(* Logix 5000 project; controller RSL5k_18_Template_noLib Emulate 5570 rev 32.11; software revision 32.02; part 15 of 16 *)
(* tags used below, declared in another part *)
   L_TaskMonitor : L_TaskMon[8];

        [450].Desc := 'Two Phases Lost In Power Cell #22', [451].Code := 351, [451].Desc := 'Bypass Failure (OV) In Power Cell #22', [452].Code := 353, [452].Desc := 'IGBT Over Current In Power Cell #23', [453].Code := 354, [453].Desc := 'Capacitor Abnormal In Power Cell #23', [454].Code := 355, [454].Desc := 'Input Over Voltage In Power Cell #23', [455].Code := 356, [455].Desc := 'DC Bus Undervoltage In Power Cell #23', [456].Code := 357, [456].Desc := 'Communication Error In Power Cell #23', [457].Code := 358, [457].Desc := 'No PWM Pulse For IGBT In Power Cell #23', [458].Code := 359, [458].Desc := 'Bypass Hardware Fault In Power Cell #23', [459].Code := 360, [459].Desc := 'Comm Link Fault in Power Cell #23', [460].Code := 361, [460].Desc := 'PCCB Ver. Incompatible In Power Cell #23', [461].Code := 362, [461].Desc := 'Power Cell #23 Bypassed', [462].Code := 363, [462].Desc := 'Over Temperature In Power Cell #23', [463].Code := 364, [463].Desc := 'Power Cell #23 Failed To Bypass', [464].Code := 365, [464].Desc := 'One Phase Lost In Power Cell #23', [465].Code := 366, [465].Desc := 'Two Phases Lost In Power Cell #23', [466].Code := 367, [466].Desc := 'Bypass Failure (OV) In Power Cell #23', [467].Code := 369, [467].Desc := 'IGBT Over Current In Power Cell #24', [468].Code := 370, [468].Desc := 'Capacitor Abnormal In Power Cell #24', [469].Code := 371, [469].Desc := 'Input Over Voltage In Power Cell #24', [470].Code := 372, [470].Desc := 'DC Bus Undervoltage In Power Cell #24', [471].Code := 373, [471].Desc := 'Communication Error In Power Cell #24', [472].Code := 374, [472].Desc := 'No PWM Pulse For IGBT In Power Cell #24', [473].Code := 375, [473].Desc := 'Bypass Hardware Fault In Power Cell #24', [474].Code := 376, [474].Desc := 'Comm Link Fault in Power Cell #24', [475].Code := 377, [475].Desc := 'PCCB Ver. Incompatible In Power Cell #24', [476].Code := 378, [476].Desc := 'Power Cell #24 Bypassed', [477].Code := 379, [477].Desc := 'Over Temperature In Power Cell #24', [478].Code := 380, [478].Desc := 'Power Cell #24 Failed To Bypass', [479].Code := 381, [479].Desc := 'One Phase Lost In Power Cell #24', [480].Code := 382,
        [480].Desc := 'Two Phases Lost In Power Cell #24', [481].Code := 383, [481].Desc := 'Bypass Failure (OV) In Power Cell #24', [482].Code := 385, [482].Desc := 'IGBT Over Current In Power Cell #25', [483].Code := 386, [483].Desc := 'Capacitor Abnormal In Power Cell #25', [484].Code := 387, [484].Desc := 'Input Over Voltage In Power Cell #25', [485].Code := 388, [485].Desc := 'DC Bus Undervoltage In Power Cell #25', [486].Code := 389, [486].Desc := 'Communication Error In Power Cell #25', [487].Code := 390, [487].Desc := 'No PWM Pulse For IGBT In Power Cell #25', [488].Code := 391, [488].Desc := 'Bypass Hardware Fault In Power Cell #25', [489].Code := 392, [489].Desc := 'Comm Link Fault in Power Cell #25', [490].Code := 393, [490].Desc := 'PCCB Ver. Incompatible In Power Cell #25', [491].Code := 394, [491].Desc := 'Power Cell #25 Bypassed', [492].Code := 395, [492].Desc := 'Over Temperature In Power Cell #25', [493].Code := 396, [493].Desc := 'Power Cell #25 Failed To Bypass', [494].Code := 397, [494].Desc := 'One Phase Lost In Power Cell #25', [495].Code := 398, [495].Desc := 'Two Phases Lost In Power Cell #25', [496].Code := 399, [496].Desc := 'Bypass Failure (OV) In Power Cell #25', [497].Code := 401, [497].Desc := 'IGBT Over Current In Power Cell #26', [498].Code := 402, [498].Desc := 'Capacitor Abnormal In Power Cell #26', [499].Code := 403, [499].Desc := 'Input Over Voltage In Power Cell #26', [500].Code := 404, [500].Desc := 'DC Bus Undervoltage In Power Cell #26', [501].Code := 405, [501].Desc := 'Communication Error In Power Cell #26', [502].Code := 406, [502].Desc := 'No PWM Pulse For IGBT In Power Cell #26', [503].Code := 407, [503].Desc := 'Bypass Hardware Fault In Power Cell #26', [504].Code := 408, [504].Desc := 'Comm Link Fault in Power Cell #26', [505].Code := 409, [505].Desc := 'PCCB Ver. Incompatible In Power Cell #26', [506].Code := 410, [506].Desc := 'Power Cell #26 Bypassed', [507].Code := 411, [507].Desc := 'Over Temperature In Power Cell #26', [508].Code := 412, [508].Desc := 'Power Cell #26 Failed To Bypass', [509].Code := 413, [509].Desc := 'One Phase Lost In Power Cell #26', [510].Code := 414,
        [510].Desc := 'Two Phases Lost In Power Cell #26', [511].Code := 415, [511].Desc := 'Bypass Failure (OV) In Power Cell #26', [512].Code := 417, [512].Desc := 'IGBT Over Current In Power Cell #27', [513].Code := 418, [513].Desc := 'Capacitor Abnormal In Power Cell #27', [514].Code := 419, [514].Desc := 'Input Over Voltage In Power Cell #27', [515].Code := 420, [515].Desc := 'DC Bus Undervoltage In Power Cell #27', [516].Code := 421, [516].Desc := 'Communication Error In Power Cell #27', [517].Code := 422, [517].Desc := 'No PWM Pulse For IGBT In Power Cell #27', [518].Code := 423, [518].Desc := 'Bypass Hardware Fault In Power Cell #27', [519].Code := 424, [519].Desc := 'Comm Link Fault in Power Cell #27', [520].Code := 425, [520].Desc := 'PCCB Ver. Incompatible In Power Cell #27', [521].Code := 426, [521].Desc := 'Power Cell #27 Bypassed', [522].Code := 427, [522].Desc := 'Over Temperature In Power Cell #27', [523].Code := 428, [523].Desc := 'Power Cell #27 Failed To Bypass', [524].Code := 429, [524].Desc := 'One Phase Lost In Power Cell #27', [525].Code := 430, [525].Desc := 'Two Phases Lost In Power Cell #27', [526].Code := 431, [526].Desc := 'Bypass Failure (OV) In Power Cell #27', [527].Code := 497, [527].Desc := 'PWMA Board Not Compatible With PCCBA1', [528].Code := 498, [528].Desc := 'PWMA Board Not Compatible With PCCBA2', [529].Code := 499, [529].Desc := 'PWMA Board Not Compatible With PCCBA3', [530].Code := 500, [530].Desc := 'PWMA Board Not Compatible With PCCBA4', [531].Code := 501, [531].Desc := 'PWMA Board Not Compatible With PCCBA5', [532].Code := 502, [532].Desc := 'PWMA Board Not Compatible With PCCBA6', [533].Code := 503, [533].Desc := 'PWMA Board Not Compatible With PCCBA7', [534].Code := 504, [534].Desc := 'PWMA Board Not Compatible With PCCBA8', [535].Code := 505, [535].Desc := 'PWMA Board Not Compatible With PCCBA9', [536].Code := 513, [536].Desc := 'PWMB Board Not Compatible With PCCBB1', [537].Code := 514, [537].Desc := 'PWMB Board Not Compatible With PCCBB2', [538].Code := 515, [538].Desc := 'PWMB Board Not Compatible With PCCBB3', [539].Code := 516, [539].Desc := 'PWMB Board Not Compatible With PCCBB4', [540].Code := 517,
        [540].Desc := 'PWMB Board Not Compatible With PCCBB5', [541].Code := 518, [541].Desc := 'PWMB Board Not Compatible With PCCBB6', [542].Code := 519, [542].Desc := 'PWMB Board Not Compatible With PCCBB7', [543].Code := 520, [543].Desc := 'PWMB Board Not Compatible With PCCBB8', [544].Code := 521, [544].Desc := 'PWMB Board Not Compatible With PCCBB9', [545].Code := 529, [545].Desc := 'PWMC Board Not Compatible With PCCBC1', [546].Code := 530, [546].Desc := 'PWMC Board Not Compatible With PCCBC2', [547].Code := 531, [547].Desc := 'PWMC Board Not Compatible With PCCBC3', [548].Code := 532, [548].Desc := 'PWMC Board Not Compatible With PCCBC4', [549].Code := 533, [549].Desc := 'PWMC Board Not Compatible With PCCBC5', [550].Code := 534, [550].Desc := 'PWMC Board Not Compatible With PCCBC6', [551].Code := 535, [551].Desc := 'PWMC Board Not Compatible With PCCBC7', [552].Code := 536, [552].Desc := 'PWMC Board Not Compatible With PCCBC8', [553].Code := 537, [553].Desc := 'PWMC Board Not Compatible With PCCBC9', [554].Code := 545, [554].Desc := 'Primary FPGA Not Compatible With PWMA', [555].Code := 546, [555].Desc := 'Primary FPGA Not Compatible With PWMB', [556].Code := 547, [556].Desc := 'Primary FPGA Not Compatible With PWMC', [557].Code := 548, [557].Desc := 'Primary FPGA Not Compatible With DT', [558].Code := 549, [558].Desc := 'Pri. DSP Not Compatible With Pri. FPGA', [559].Code := 550, [559].Desc := 'Pri. DSP Not Compatible With Sec. DSP', [560].Code := 553, [560].Desc := 'Primary DSP Not Compatible With PLC', [561].Code := 673, [561].Desc := 'User Defined Fault #1', [562].Code := 674, [562].Desc := 'User Defined Fault #2', [563].Code := 675, [563].Desc := 'User Defined Fault #3', [564].Code := 676, [564].Desc := 'User Defined Fault #4', [565].Code := 677, [565].Desc := 'User Defined Fault #5', [566].Code := 678, [566].Desc := 'User Defined Fault #6', [567].Code := 679, [567].Desc := 'User Defined Fault #7', [568].Code := 680, [568].Desc := 'User Defined Fault #8', [569].Code := 681, [569].Desc := 'User Defined Fault #9', [570].Code := 682,
        [570].Desc := 'User Defined Fault #10', [571].Code := 683, [571].Desc := 'User Defined Fault #11', [572].Code := 684, [572].Desc := 'User Defined Fault #12', [573].Code := 685, [573].Desc := 'User Defined Fault #13', [574].Code := 686, [574].Desc := 'User Defined Fault #14', [575].Code := 687, [575].Desc := 'User Defined Fault #15', [576].Code := 688, [576].Desc := 'User Defined Fault #16', [577].Code := 689, [577].Desc := 'User Defined Warning #1', [578].Code := 690, [578].Desc := 'User Defined Warning #2', [579].Code := 691, [579].Desc := 'User Defined Warning #3', [580].Code := 692, [580].Desc := 'User Defined Warning #4', [581].Code := 693, [581].Desc := 'User Defined Warning #5', [582].Code := 694, [582].Desc := 'User Defined Warning #6', [583].Code := 695, [583].Desc := 'User Defined Warning #7', [584].Code := 696, [584].Desc := 'User Defined Warning #8', [585].Code := 697, [585].Desc := 'User Defined Warning #9', [586].Code := 698, [586].Desc := 'User Defined Warning #10', [587].Code := 699, [587].Desc := 'User Defined Warning #11', [588].Code := 700, [588].Desc := 'User Defined Warning #12', [589].Code := 701, [589].Desc := 'User Defined Warning #13', [590].Code := 702, [590].Desc := 'User Defined Warning #14', [591].Code := 703, [591].Desc := 'User Defined Warning #15', [592].Code := 704, [592].Desc := 'User Defined Warning #16');   // PowerFlex 6000 MV VFD FW6.x Fault Codes and Descriptions
   PF7000_FaultCodeList : P_DescList[500];   // PowerFlex 7000 MV VFD Fault Codes and Descriptions
   PF700S_FaultCodeList : P_DescList[80] := ([0].Desc := 'Check drive manual for this fault code', [1].Code := 48, [1].Desc := 'No Controlling Device', [2].Code := 49, [2].Desc := 'DPI Loss Port 1', [3].Code := 50, [3].Desc := 'DPI Loss Port 2', [4].Code := 51, [4].Desc := 'DPI Loss Port 3', [5].Code := 52, [5].Desc := 'DPI Loss Port 4', [6].Code := 53, [6].Desc := 'DPI Loss Port 5', [7].Code := 54, [7].Desc := 'DPI Loss Port 6', [8].Code := 55, [8].Desc := 'Network Loss DPI Port 1', [9].Code := 56, [9].Desc := 'Network Loss DPI Port 2', [10].Code := 57, [10].Desc := 'Network Loss DPI Port 3', [11].Code := 58, [11].Desc := 'Network Loss DPI Port 4', [12].Code := 59, [12].Desc := 'Network Loss DPI Port 5', [13].Code := 60, [13].Desc := 'Network Loss DPI Port 6', [14].Code := 9, [14].Desc := 'SyncLink Communication Fault', [15].Code := 10, [15].Desc := 'Drive Power Loss', [16].Code := 11, [16].Desc := 'Motor Overload Tripped', [17].Code := 12, [17].Desc := 'Motor Overload Pending', [18].Code := 27, [18].Desc := 'Instantaneous Motor Overcurrent', [19].Code := 26, [19].Desc := 'Ground Fault', [20].Code := 18, [20].Desc := 'External Fault Input', [21].Code := 1, [21].Desc := 'Absolute Overspeed Detected', [22].Code := 2, [22].Desc := 'Vref Deceleration Failed', [23].Code := 3, [23].Desc := 'Encoder 0 Loss', [24].Code := 4, [24].Desc := 'Encoder 1 Loss', [25].Code := 5, [25].Desc := 'Option Port 0 Loss', [26].Code := 6, [26].Desc := 'Option Port 1 Loss', [27].Code := 13, [27].Desc := 'Motor Stalled', [28].Code := 14, [28].Desc := 'Inverter Overtemperature Pending', [29].Code := 15, [29].Desc := 'Inverter Overtemperature Trip', [30].Code := 16,
        [30].Desc := 'Inverter Overload Pending', [31].Code := 17, [31].Desc := 'Inverter Overload Trip', [32].Code := 19, [32].Desc := 'DSP Memory Error', [33].Code := 20, [33].Desc := 'DSP Device Error', [34].Code := 21, [34].Desc := 'Error Inertia Test', [35].Code := 22, [35].Desc := 'Overfrequency Fault', [36].Code := 23, [36].Desc := 'MC Commissioning Failed', [37].Code := 24, [37].Desc := 'DC Bus Overvoltage', [38].Code := 28, [38].Desc := 'VPL/MC Communication Fail', [39].Code := 29, [39].Desc := 'PWM Signal Short', [40].Code := 30, [40].Desc := 'MC Firmware Fault', [41].Code := 31, [41].Desc := 'Precharge Error', [42].Code := 32, [42].Desc := 'PWM Not Synchronized', [43].Code := 33, [43].Desc := '+/- 12V Power Fault', [44].Code := 35, [44].Desc := 'Controller EEPROM Checksum', [45].Code := 38, [45].Desc := 'Brake Overload Trip', [46].Code := 39, [46].Desc := 'Power EEPROM CRC Failed', [47].Code := 40, [47].Desc := 'SyncLink Multiplier Overflow', [48].Code := 41, [48].Desc := 'Bus Loss Ridethru Timed Out', [49].Code := 42, [49].Desc := 'DC Bus Undervoltage', [50].Code := 43, [50].Desc := 'Voltage Feedback Loss', [51].Code := 44, [51].Desc := 'Runtime Data were Reset', [52].Code := 46, [52].Desc := 'Interpolator Out of Sync', [53].Code := 61, [53].Desc := 'DriveLogix Taken Out of Run Mode', [54].Code := 62, [54].Desc := 'DriveLogix Communication Timeout', [55].Code := 63, [55].Desc := 'DriveLogix Connection Closed', [56].Code := 64, [56].Desc := 'DriveLogix Comm Format Changed', [57].Code := 65, [57].Desc := 'HiHP Drive: Input AC Phase Loss', [58].Code := 66, [58].Desc := 'HiHP Drive: Bus Communication Delay', [59].Code := 67, [59].Desc := 'HiHP Drive: Bus Comm Link Loss', [60].Code := 68,
        [60].Desc := 'HiHP Drive: Bus CRC Error', [61].Code := 69, [61].Desc := 'HiHP Drive: Bus Watchdog Timeout', [62].Code := 70, [62].Desc := 'HiHP Drive: Fan Feedback Lost', [63].Code := 71, [63].Desc := 'HiHP Drive: Overload', [64].Code := 72, [64].Desc := 'HiHP Drive: Power Board Proc Error', [65].Code := 73, [65].Desc := 'HiHP Drive: Precharge Contactor Fault', [66].Code := 74, [66].Desc := 'HiHP Drive: Power EEPROM Error', [67].Code := 75, [67].Desc := 'HiHP Drive: Power Board Overtemp', [68].Code := 85, [68].Desc := 'Position Error');   // PowerFlex 700S VFD Fault Codes and Descriptions
   PF75x_FaultCodeList : P_DescList[212] := ([0].Desc := 'Check drive manual for this fault code', [1].Code := 13032, [1].Desc := 'I/O Network Communication Fault', [2].Code := 13035, [2].Desc := 'I/O Network Idle (Controller in PROG)', [3].Code := 13030, [3].Desc := 'I/O Network Link Removed', [4].Code := 13031, [4].Desc := 'I/O Network Duplicate Address', [5].Code := 13033, [5].Desc := 'I/O Network Sent Reset Command', [6].Code := 13034, [6].Desc := 'I/O Network Connection Closed', [7].Code := 13037, [7].Desc := 'I/O Network Timed Out', [8].Code := 13044, [8].Desc := 'Control Network Message Timed Out', [9].Code := 13046, [9].Desc := 'Peer-to-Peer I/O Timed Out', [10].Code := 13056, [10].Desc := 'Drive Could Not Send e-mail', [11].Code := 13057, [11].Desc := 'I/O Network Adapter Fault', [12].Code := 13058, [12].Desc := 'I/O Network Adapter Set to Defaults', [13].Code := 2, [13].Desc := 'Auxiliary Input Interlock', [14].Code := 3, [14].Desc := 'Power Failure', [15].Code := 4, [15].Desc := 'Bus Undervoltage', [16].Code := 5, [16].Desc := 'Bus Overvoltage', [17].Code := 7, [17].Desc := 'Motor Overload', [18].Code := 8, [18].Desc := 'Heatsink Overtemperature', [19].Code := 9, [19].Desc := 'Transistor Overtemperature', [20].Code := 10, [20].Desc := 'Dynamic Brake Resistor Overtemperature', [21].Code := 12, [21].Desc := 'Hardware Overcurrent', [22].Code := 13, [22].Desc := 'Ground Fault', [23].Code := 14, [23].Desc := 'Ground Warning', [24].Code := 15, [24].Desc := 'Load Loss', [25].Code := 17, [25].Desc := 'Input Phase Loss', [26].Code := 18, [26].Desc := 'Motor Pos. Temp. Coeff. Trip', [27].Code := 20, [27].Desc := 'Torque Prv. Speed Band Fault', [28].Code := 21, [28].Desc := 'Output Phase Loss', [29].Code := 24, [29].Desc := 'Deceleration Inhibited', [30].Code := 25,
        [30].Desc := 'Over Speed Limit', [31].Code := 29, [31].Desc := 'Analog Input Signal Loss', [32].Code := 33, [32].Desc := 'Auto Restart Tries Exhausted', [33].Code := 36, [33].Desc := 'Output Current Over Rating', [34].Code := 38, [34].Desc := 'Phase U Ground Fault', [35].Code := 39, [35].Desc := 'Phase V Ground Fault', [36].Code := 40, [36].Desc := 'Phase W Ground Fault', [37].Code := 41, [37].Desc := 'Phase U to V Shorted', [38].Code := 42, [38].Desc := 'Phase V to W Shorted', [39].Code := 43, [39].Desc := 'Phase W to U Shorted', [40].Code := 44, [40].Desc := 'Phase U (Neg) Ground Fault', [41].Code := 45, [41].Desc := 'Phase V (Neg) Ground Fault', [42].Code := 46, [42].Desc := 'Phase W (Neg) Ground Fault', [43].Code := 48, [43].Desc := 'Drive Set to Default Configuration', [44].Code := 55, [44].Desc := 'Drive Control Board Overtemperature', [45].Code := 58, [45].Desc := 'Drive Module Set to Default Values', [46].Code := 61, [46].Desc := 'Shear Pin (1)', [47].Code := 62, [47].Desc := 'Shear Pin (2)', [48].Code := 64, [48].Desc := 'Drive OverLoad', [49].Code := 71, [49].Desc := 'Port 1 Adapter Fault', [50].Code := 72, [50].Desc := 'Port 2 Adapter Fault', [51].Code := 73, [51].Desc := 'Port 3 Adapter Fault', [52].Code := 74, [52].Desc := 'Port 4 Adapter Fault', [53].Code := 75, [53].Desc := 'Port 5 Adapter Fault', [54].Code := 76, [54].Desc := 'Port 6 Adapter Fault', [55].Code := 77, [55].Desc := 'IR Volts Range', [56].Code := 78, [56].Desc := 'Flux Amps Reference Rating', [57].Code := 79, [57].Desc := 'Excessive Load', [58].Code := 80, [58].Desc := 'Drive Autotune Aborted', [59].Code := 81, [59].Desc := 'Port 1 DPI Communication Loss', [60].Code := 82,
        [60].Desc := 'Port 2 DPI Communication Loss', [61].Code := 83, [61].Desc := 'Port 3 DPI Communication Loss', [62].Code := 84, [62].Desc := 'Port 4 DPI Communication Loss', [63].Code := 85, [63].Desc := 'Port 5 DPI Communication Loss', [64].Code := 86, [64].Desc := 'Port 6 DPI Communication Loss', [65].Code := 87, [65].Desc := 'IXo Voltage Range', [66].Code := 91, [66].Desc := 'Primary Velocity Feedback Lost', [67].Code := 93, [67].Desc := 'Hardware Enable Jumper Problem', [68].Code := 94, [68].Desc := 'Alternate Velocity Feedback Lost', [69].Code := 95, [69].Desc := 'Auxiliary Velocity Feedback Lost', [70].Code := 96, [70].Desc := 'Position Feedback Lost', [71].Code := 97, [71].Desc := 'Auto Tach Switch Failure', [72].Code := 137, [72].Desc := 'External Precharge Error', [73].Code := 138, [73].Desc := 'Precharge Open', [74].Code := 152, [74].Desc := 'No Source Defined for Stop Command', [75].Code := 168, [75].Desc := 'Heatsink Undertemp (sensor fail)', [76].Code := 175, [76].Desc := 'Travel Limits Conflicting', [77].Code := 181, [77].Desc := 'Reached Forward End of Travel', [78].Code := 182, [78].Desc := 'Reached Reverse End of Travel', [79].Code := 203, [79].Desc := 'Port 13 Adapter (Ethernet) Fault', [80].Code := 204, [80].Desc := 'Port 14 Adapter (DriveLogix) Fault', [81].Code := 210, [81].Desc := 'Safety Option Enable Jumper is Out', [82].Code := 211, [82].Desc := 'Safety Option Board Fault', [83].Code := 212, [83].Desc := 'Safety Jumper Not Present', [84].Code := 213, [84].Desc := 'Safety Jumper Needs Removed', [85].Code := 224, [85].Desc := 'Port 4 Communication Lost', [86].Code := 225, [86].Desc := 'Port 5 Communication Lost', [87].Code := 226, [87].Desc := 'Port 6 Communication Lost', [88].Code := 227, [88].Desc := 'Port 7 Communication Lost', [89].Code := 228, [89].Desc := 'Port 8 Communication Lost', [90].Code := 229,
        [90].Desc := 'Port 9 Communication Lost', [91].Code := 230, [91].Desc := 'Port 10 Communication Lost', [92].Code := 231, [92].Desc := 'Port 11 Communication Lost', [93].Code := 232, [93].Desc := 'Port 12 Communication Lost', [94].Code := 233, [94].Desc := 'Port 13 Communication Lost', [95].Code := 234, [95].Desc := 'Port 14 Communication Lost', [96].Code := 315, [96].Desc := 'Excess Position Error', [97].Code := 331, [97].Desc := 'Inverter Board I1 Communication Failed', [98].Code := 332, [98].Desc := 'Inverter Board I2 Communication Failed', [99].Code := 341, [99].Desc := 'Converter Board C1 Communication Failed', [100].Code := 342, [100].Desc := 'Converter Board C2 Communication Failed', [101].Code := 371, [101].Desc := 'Precharge Board P1 Communication Failed', [102].Code := 372, [102].Desc := 'Precharge Board P2 Communication Failed', [103].Code := 918, [103].Desc := 'Control Task Overload', [104].Code := 919, [104].Desc := 'System Task Overload', [105].Code := 920, [105].Desc := '5 millisecond Task Overload', [106].Code := 10101, [106].Desc := 'Inverter I1 Communication Failed', [107].Code := 10104, [107].Desc := 'Inverter I1 U+ Phase Overcurrent', [108].Code := 10105, [108].Desc := 'Inverter I1 U- Phase Overcurrent', [109].Code := 10106, [109].Desc := 'Inverter I1 V+ Phase Overcurrent', [110].Code := 10107, [110].Desc := 'Inverter I1 V- Phase Overcurrent', [111].Code := 10108, [111].Desc := 'Inverter I1 W+ Phase Overcurrent', [112].Code := 10109, [112].Desc := 'Inverter I1 W- Phase Overcurrent', [113].Code := 10110, [113].Desc := 'Inverter I1 Bus Overvoltage', [114].Code := 10111, [114].Desc := 'Inverter I1 Ground Fault', [115].Code := 10112, [115].Desc := 'Inverter I1 IGBT Overtemperature', [116].Code := 10113, [116].Desc := 'Inverter I1 Heatsink Overtemperature', [117].Code := 10114, [117].Desc := 'Inverter I1 Main Power Low', [118].Code := 10115, [118].Desc := 'Inverter I1 Interface Power Low', [119].Code := 10117, [119].Desc := 'Inverter I1 System Power Overcurrent', [120].Code := 10120,
        [120].Desc := 'Inverter I1 PLI Board Overtemperature', [121].Code := 10121, [121].Desc := 'Inverter I1 PS Board Overtemperature', [122].Code := 10129, [122].Desc := 'Inverter I1 DC Bus Imbalance', [123].Code := 10134, [123].Desc := 'Inverter I1 Phase U Gate Board Fault', [124].Code := 10135, [124].Desc := 'Inverter I1 Phase V Gate Board Fault', [125].Code := 10136, [125].Desc := 'Inverter I1 Phase W Gate Board Fault', [126].Code := 10201, [126].Desc := 'Inverter I2 Communication Failed', [127].Code := 10204, [127].Desc := 'Inverter I2 U+ Phase Overcurrent', [128].Code := 10205, [128].Desc := 'Inverter I2 U- Phase Overcurrent', [129].Code := 10206, [129].Desc := 'Inverter I2 V+ Phase Overcurrent', [130].Code := 10207, [130].Desc := 'Inverter I2 V- Phase Overcurrent', [131].Code := 10208, [131].Desc := 'Inverter I2 W+ Phase Overcurrent', [132].Code := 10209, [132].Desc := 'Inverter I2 W- Phase Overcurrent', [133].Code := 10210, [133].Desc := 'Inverter I2 Bus Overvoltage', [134].Code := 10211, [134].Desc := 'Inverter I2 Ground Fault', [135].Code := 10212, [135].Desc := 'Inverter I2 IGBT Overtemperature', [136].Code := 10213, [136].Desc := 'Inverter I2 Heatsink Overtemperature', [137].Code := 10214, [137].Desc := 'Inverter I2 Main Power Low', [138].Code := 10215, [138].Desc := 'Inverter I2 Interface Power Low', [139].Code := 10217, [139].Desc := 'Inverter I2 System Power Overcurrent', [140].Code := 10220, [140].Desc := 'Inverter I2 PLI Board Overtemperature', [141].Code := 10221, [141].Desc := 'Inverter I2 PS Board Overtemperature', [142].Code := 10229, [142].Desc := 'Inverter I2 DC Bus Imbalance', [143].Code := 10234, [143].Desc := 'Inverter I2 Phase U Gate Board Fault', [144].Code := 10235, [144].Desc := 'Inverter I2 Phase V Gate Board Fault', [145].Code := 10236, [145].Desc := 'Inverter I2 Phase W Gate Board Fault', [146].Code := 10301, [146].Desc := 'Inverter I3 Communication Failed', [147].Code := 10304, [147].Desc := 'Inverter I3 U+ Phase Overcurrent', [148].Code := 10305, [148].Desc := 'Inverter I3 U- Phase Overcurrent', [149].Code := 10306, [149].Desc := 'Inverter I3 V+ Phase Overcurrent', [150].Code := 10307,
        [150].Desc := 'Inverter I3 V- Phase Overcurrent', [151].Code := 10308, [151].Desc := 'Inverter I3 W+ Phase Overcurrent', [152].Code := 10309, [152].Desc := 'Inverter I3 W- Phase Overcurrent', [153].Code := 10310, [153].Desc := 'Inverter I3 Bus Overvoltage', [154].Code := 10311, [154].Desc := 'Inverter I3 Ground Fault', [155].Code := 10312, [155].Desc := 'Inverter I3 IGBT Overtemperature', [156].Code := 10313, [156].Desc := 'Inverter I3 Heatsink Overtemperature', [157].Code := 10314, [157].Desc := 'Inverter I3 Main Power Low', [158].Code := 10315, [158].Desc := 'Inverter I3 Interface Power Low', [159].Code := 10317, [159].Desc := 'Inverter I3 System Power Overcurrent', [160].Code := 10320, [160].Desc := 'Inverter I3 PLI Board Overtemperature', [161].Code := 10321, [161].Desc := 'Inverter I3 PS Board Overtemperature', [162].Code := 10329, [162].Desc := 'Inverter I3 DC Bus Imbalance', [163].Code := 10334, [163].Desc := 'Inverter I3 Phase U Gate Board Fault', [164].Code := 10335, [164].Desc := 'Inverter I3 Phase V Gate Board Fault', [165].Code := 10336, [165].Desc := 'Inverter I3 Phase W Gate Board Fault', [166].Code := 11101, [166].Desc := 'Converter C1 Precharge Problem', [167].Code := 11111, [167].Desc := 'Converter C1 SCR Overtemperature', [168].Code := 11112, [168].Desc := 'Converter C1 Heat Sink Overtemp', [169].Code := 11115, [169].Desc := 'Converter C1 Line/Bus Voltage Dip', [170].Code := 11117, [170].Desc := 'Converter C1 Line Frequency Fault', [171].Code := 11118, [171].Desc := 'Converter C1 Single Phase Fault', [172].Code := 11134, [172].Desc := 'Converter C1 Overcurrent', [173].Code := 11135, [173].Desc := 'Converter C1 Ground Fault', [174].Code := 11138, [174].Desc := 'Converter C1 Board Overtemperature', [175].Code := 11141, [175].Desc := 'Converter C1 DC Power Supply Fault', [176].Code := 11142, [176].Desc := 'Converter C1 Communication Lost', [177].Code := 11160, [177].Desc := 'Converter C1 Bus Asymmetry Stop', [178].Code := 11161, [178].Desc := 'Converter C1 AC Line Overvoltage', [179].Code := 11162, [179].Desc := 'Converter C1 AC Line Lost', [180].Code := 11163,
        [180].Desc := 'Converter C1 Fault Queue Full', [181].Code := 11201, [181].Desc := 'Converter C2 Precharge Problem', [182].Code := 11211, [182].Desc := 'Converter C2 SCR Overtemperature', [183].Code := 11212, [183].Desc := 'Converter C2 Heat Sink Overtemp', [184].Code := 11215, [184].Desc := 'Converter C2 Line/Bus Voltage Dip', [185].Code := 11217, [185].Desc := 'Converter C2 Line Frequency Fault', [186].Code := 11218, [186].Desc := 'Converter C2 Single Phase Fault', [187].Code := 11234, [187].Desc := 'Converter C2 Overcurrent', [188].Code := 11235, [188].Desc := 'Converter C2 Ground Fault', [189].Code := 11238, [189].Desc := 'Converter C2 Board Overtemperature', [190].Code := 11241, [190].Desc := 'Converter C2 DC Power Supply Fault', [191].Code := 11242, [191].Desc := 'Converter C2 Communication Lost', [192].Code := 11260, [192].Desc := 'Converter C2 Bus Asymmetry Stop', [193].Code := 11261, [193].Desc := 'Converter C2 AC Line Overvoltage', [194].Code := 11262, [194].Desc := 'Converter C2 AC Line Lost', [195].Code := 11263, [195].Desc := 'Converter C2 Fault Queue Full', [196].Code := 11201, [196].Desc := 'Converter C2 Precharge Problem', [197].Code := 11211, [197].Desc := 'Converter C2 SCR Overtemperature', [198].Code := 11212, [198].Desc := 'Converter C2 Heat Sink Overtemp', [199].Code := 11215, [199].Desc := 'Converter C2 Line/Bus Voltage Dip', [200].Code := 11217, [200].Desc := 'Converter C2 Line Frequency Fault', [201].Code := 11218, [201].Desc := 'Converter C2 Single Phase Fault', [202].Code := 11234, [202].Desc := 'Converter C2 Overcurrent', [203].Code := 11235, [203].Desc := 'Converter C2 Ground Fault', [204].Code := 11238, [204].Desc := 'Converter C2 Board Overtemperature', [205].Code := 11241, [205].Desc := 'Converter C2 DC Power Supply Fault', [206].Code := 11242, [206].Desc := 'Converter C2 Communication Lost', [207].Code := 11260, [207].Desc := 'Converter C2 Bus Asymmetry Stop', [208].Code := 11261, [208].Desc := 'Converter C2 AC Line Overvoltage', [209].Code := 11262, [209].Desc := 'Converter C2 AC Line Lost', [210].Code := 11263,
        [210].Desc := 'Converter C2 Fault Queue Full');   // PowerFlex 753 / 755 Fault Codes and Descriptions
   PF7xx_FaultCodeList : P_DescList[120] := ([0].Desc := 'Check drive manual for this fault code', [1].Code := 121, [1].Desc := 'I/O Communication Loss', [2].Code := 122, [2].Desc := 'I/O Failure', [3].Code := 91, [3].Desc := 'Encoder Loss', [4].Code := 92, [4].Desc := 'Pulse Input Loss', [5].Code := 93, [5].Desc := 'Hardware Fault', [6].Code := 94, [6].Desc := 'Hardware Enable Missing', [7].Code := 1, [7].Desc := 'Precharge Active', [8].Code := 2, [8].Desc := 'Auxiliary Input', [9].Code := 3, [9].Desc := 'Power Loss', [10].Code := 4, [10].Desc := 'Under Voltage', [11].Code := 5, [11].Desc := 'Over Voltage', [12].Code := 6, [12].Desc := 'Motor Stall', [13].Code := 7, [13].Desc := 'Motor Overload', [14].Code := 8, [14].Desc := 'Heatsink OverTemp', [15].Code := 9, [15].Desc := 'IGBT OverTemp', [16].Code := 10, [16].Desc := 'System Fault', [17].Code := 12, [17].Desc := 'Hardware Overcurrent', [18].Code := 13, [18].Desc := 'Ground Fault', [19].Code := 14, [19].Desc := 'Inverter Fault', [20].Code := 15, [20].Desc := 'Load Loss', [21].Code := 16, [21].Desc := 'Motor Thermistor', [22].Code := 17, [22].Desc := 'Input Phase Loss', [23].Code := 19, [23].Desc := 'Unbalanced Power', [24].Code := 20, [24].Desc := 'Torque Prover Speed Band', [25].Code := 21, [25].Desc := 'Output Phase Loss', [26].Code := 22, [26].Desc := 'Nameplate Hz Conflict', [27].Code := 23, [27].Desc := 'Max Frequency Conflict', [28].Code := 24, [28].Desc := 'Decel Inhibit', [29].Code := 25, [29].Desc := 'Over Speed Limit', [30].Code := 26,
        [30].Desc := 'VHz Negative Slope', [31].Code := 27, [31].Desc := 'Speed Reference Conflict', [32].Code := 28, [32].Desc := 'Braking Resistor Missing', [33].Code := 29, [33].Desc := 'Analog Input Loss', [34].Code := 31, [34].Desc := 'IGBT Temperature HW', [35].Code := 32, [35].Desc := 'Fan Cooling Fault', [36].Code := 33, [36].Desc := 'Auto Restart Tries', [37].Code := 34, [37].Desc := 'CAN Bus Fault', [38].Code := 36, [38].Desc := 'Software Overcurrent', [39].Code := 37, [39].Desc := 'Heatsink Under Temperature', [40].Code := 38, [40].Desc := 'Phase U to Ground', [41].Code := 39, [41].Desc := 'Phase V to Ground', [42].Code := 40, [42].Desc := 'Phase W to Ground', [43].Code := 41, [43].Desc := 'Phase U-V Short', [44].Code := 42, [44].Desc := 'Phase U-W Short', [45].Code := 43, [45].Desc := 'Phase V-W Short', [46].Code := 44, [46].Desc := 'Device Changed', [47].Code := 45, [47].Desc := 'Device Added', [48].Code := 47, [48].Desc := 'NVS Read Checksum', [49].Code := 48, [49].Desc := 'Params Defaulted', [50].Code := 48, [50].Desc := 'Params Defaulted', [51].Code := 49, [51].Desc := 'Drive Powerup', [52].Code := 51, [52].Desc := 'Fault Queue Cleared', [53].Code := 52, [53].Desc := 'Faults Cleared', [54].Code := 55, [54].Desc := 'Control Board Overtemp', [55].Code := 59, [55].Desc := 'Gate Disable', [56].Code := 60, [56].Desc := 'Hardware Thermistor', [57].Code := 63, [57].Desc := 'Shear Pin', [58].Code := 64, [58].Desc := 'Drive Overload', [59].Code := 65, [59].Desc := 'I/O Removed', [60].Code := 69,
        [60].Desc := 'D B Resistance', [61].Code := 70, [61].Desc := 'Power Unit Fault', [62].Code := 71, [62].Desc := 'Port 1 Adapter', [63].Code := 72, [63].Desc := 'Port 2 Adapter', [64].Code := 73, [64].Desc := 'Port 3 Adapter', [65].Code := 74, [65].Desc := 'Port 4 Adapter', [66].Code := 75, [66].Desc := 'Port 5 Adapter', [67].Code := 76, [67].Desc := 'Port 6 Adapter', [68].Code := 77, [68].Desc := 'IR Volts Range', [69].Code := 78, [69].Desc := 'Flux Amps Ref Range', [70].Code := 79, [70].Desc := 'Excessive Load', [71].Code := 80, [71].Desc := 'AutoTune Aborted', [72].Code := 81, [72].Desc := 'Port 1 DPI Loss', [73].Code := 82, [73].Desc := 'Port 2 DPI Loss', [74].Code := 83, [74].Desc := 'Port 3 DPI Loss', [75].Code := 84, [75].Desc := 'Port 4 DPI Loss', [76].Code := 85, [76].Desc := 'Port 5 DPI Loss', [77].Code := 86, [77].Desc := 'Port 6 DPI Loss', [78].Code := 87, [78].Desc := 'IXo Voltage Range', [79].Code := 88, [79].Desc := 'Software Fault', [80].Code := 89, [80].Desc := 'Software Fault', [81].Code := 90, [81].Desc := 'Encoder Quad Error', [82].Code := 95, [82].Desc := 'AutoTune Rs Static Test Fail', [83].Code := 96, [83].Desc := 'AutoTune Rm Rotate Test Fail', [84].Code := 97, [84].Desc := 'AutoTune Mag Cur Rotate Test Fail', [85].Code := 98, [85].Desc := 'AutoTune Saturation Curve Test Fail', [86].Code := 99, [86].Desc := 'User Set Timed Out', [87].Code := 100, [87].Desc := 'Parameter Checksum', [88].Code := 101, [88].Desc := 'UserSet1 Checksum', [89].Code := 102, [89].Desc := 'UserSet2 Checksum', [90].Code := 103,
        [90].Desc := 'UserSet3 Checksum', [91].Code := 104, [91].Desc := 'Power Board Checksum 1', [92].Code := 105, [92].Desc := 'Power Board Checksum 2', [93].Code := 106, [93].Desc := 'Incompat. MCB-PB', [94].Code := 107, [94].Desc := 'Replaced MCB-PB', [95].Code := 108, [95].Desc := 'Analog Cal Checksum', [96].Code := 112, [96].Desc := 'Power Down Checksum', [97].Code := 113, [97].Desc := 'Fatal Application Error', [98].Code := 114, [98].Desc := 'AutoTune Enabled but Not Started', [99].Code := 120, [99].Desc := 'I/O Board Replaced', [100].Code := 130, [100].Desc := 'Hardware Fault', [101].Code := 131, [101].Desc := 'Hardware Fault', [102].Code := 133, [102].Desc := 'Digital Input Conflict A', [103].Code := 134, [103].Desc := 'Digital Input Conflict B', [104].Code := 135, [104].Desc := 'Digital Input Conflict C', [105].Code := 136, [105].Desc := 'Bipolar Conflict', [106].Code := 139, [106].Desc := 'User Set Conflict', [107].Code := 143, [107].Desc := 'TB Man Ref Select Conflict', [108].Code := 147, [108].Desc := 'Starting at Powerup', [109].Code := 148, [109].Desc := 'Internal DB Regulator Overheated', [110].Code := 149, [110].Desc := 'Wake Timer is Timing', [111].Code := 150, [111].Desc := 'Sleep Configuration Error');   // PowerFlex 70 / 700 / 700H Fault Codes and Descriptions
   PFDC_FaultCodeList : P_DescList[50] := ([0].Desc := 'Check drive manual for this fault code', [1].Code := 71, [1].Desc := 'Port 1 Adapter', [2].Code := 72, [2].Desc := 'Port 2 Adapter', [3].Code := 73, [3].Desc := 'Port 3 Adapter', [4].Code := 74, [4].Desc := 'Port 4 Adapter', [5].Code := 75, [5].Desc := 'Port 5 Adapter', [6].Code := 81, [6].Desc := 'Port 1 DPI Loss', [7].Code := 82, [7].Desc := 'Port 2 DPI Loss', [8].Code := 83, [8].Desc := 'Port 3 DPI Loss', [9].Code := 84, [9].Desc := 'Port 4 DPI Loss', [10].Code := 85, [10].Desc := 'Port 5 DPI Loss', [11].Code := 2, [11].Desc := 'Auxiliary Input', [12].Code := 3, [12].Desc := 'Power Failure', [13].Code := 4, [13].Desc := 'AC Undervoltage', [14].Code := 5, [14].Desc := 'Arm Overvoltage', [15].Code := 6, [15].Desc := 'Field Current Loss', [16].Code := 7, [16].Desc := 'Motor Overload', [17].Code := 8, [17].Desc := 'Heatsink Overtemp', [18].Code := 10, [18].Desc := 'Main Contactor', [19].Code := 13, [19].Desc := 'Overcurrent', [20].Code := 16, [20].Desc := 'Motor Overtemp', [21].Code := 25, [21].Desc := 'Overspeed', [22].Code := 37, [22].Desc := 'Inverting Fault', [23].Code := 48, [23].Desc := 'Parameters Defaulted', [24].Code := 56, [24].Desc := 'STune Overspeed', [25].Code := 57, [25].Desc := 'STune Stalled', [26].Code := 58, [26].Desc := 'STune Load Hi', [27].Code := 59, [27].Desc := 'STune Current Limit', [28].Code := 60, [28].Desc := 'STune Friction Lo', [29].Code := 61, [29].Desc := 'STune Timeout', [30].Code := 62,
        [30].Desc := 'STune Aborted', [31].Code := 64, [31].Desc := 'Drive Overload', [32].Code := 70, [32].Desc := 'Sustained Current', [33].Code := 91, [33].Desc := 'Speed Fdbk Loss', [34].Code := 92, [34].Desc := 'Encoder Error', [35].Code := 93, [35].Desc := 'Resolver Error', [36].Code := 100, [36].Desc := 'EEPROM Error', [37].Code := 130, [37].Desc := 'Hardware Fault', [38].Code := 131, [38].Desc := 'Interrupt Error', [39].Code := 132, [39].Desc := 'DSP Error');   // PowerFlex DC Drive Fault Codes and Descriptions
   SMC50_FaultCodeList : P_DescList[68] := ([0].Desc := 'Check starter manual for this fault code', [1].Code := 1, [1].Desc := 'Line Loss Phase A', [2].Code := 2, [2].Desc := 'Line Loss Phase B', [3].Code := 3, [3].Desc := 'Line Loss Phase C', [4].Code := 4, [4].Desc := 'Shorted SCR Phase A', [5].Code := 5, [5].Desc := 'Shorted SCR Phase B', [6].Code := 6, [6].Desc := 'Shorted SCR Phase C', [7].Code := 7, [7].Desc := 'Open SCR Gate Phase A', [8].Code := 8, [8].Desc := 'Open SCR Gate Phase B', [9].Code := 9, [9].Desc := 'Open SCR Gate Phase C', [10].Code := 10, [10].Desc := 'SMC-50 SCR Overtemperature', [11].Code := 14, [11].Desc := 'No Load or Load Connection Failed', [12].Code := 15, [12].Desc := 'Open Load Circuit Phase A', [13].Code := 16, [13].Desc := 'Open Load Circuit Phase B', [14].Code := 17, [14].Desc := 'Open Load Circuit Phase C', [15].Code := 18, [15].Desc := 'Voltage Imbalance', [16].Code := 19, [16].Desc := 'Line Overvoltage', [17].Code := 20, [17].Desc := 'Line Undervoltage', [18].Code := 21, [18].Desc := 'Motor Overload Trip', [19].Code := 22, [19].Desc := 'Motor Underload Trip', [20].Code := 23, [20].Desc := 'Motor / Shaft / Part Jam Trip', [21].Code := 24, [21].Desc := 'Motor Stall Trip', [22].Code := 25, [22].Desc := 'Incoming Power Phase Reversal', [23].Code := 26, [23].Desc := 'Required Expansion Module Removed', [24].Code := 27, [24].Desc := 'Expansion Module Is Incompatible', [25].Code := 28, [25].Desc := 'Expansion Module or Peripheral Fault', [26].Code := 29, [26].Desc := 'Too many motor starts in the last hour', [27].Code := 30, [27].Desc := 'Current Transformer Loss Phase A', [28].Code := 31, [28].Desc := 'Current Transformer Loss Phase B', [29].Code := 32, [29].Desc := 'Current Transformer Loss Phase C', [30].Code := 33,
        [30].Desc := 'HAL ID Fault (Incompatible Power Pole)', [31].Code := 34, [31].Desc := 'Nonvolatile (FLASH) Memory Fault', [32].Code := 36, [32].Desc := '24 VDC Control Power Supply Failure', [33].Code := 37, [33].Desc := 'Control Voltage Out of Specification', [34].Code := 38, [34].Desc := 'Configurable Fault Input #1 Triggered', [35].Code := 39, [35].Desc := 'Configurable Fault Input #2 Triggered', [36].Code := 40, [36].Desc := 'Configurable Fault Input #3 Triggered', [37].Code := 41, [37].Desc := 'Configurable Fault Input #4 Triggered', [38].Code := 42, [38].Desc := 'High Motor Current Imbalance', [39].Code := 43, [39].Desc := 'Real Power Below Configured Low Limit', [40].Code := 44, [40].Desc := 'Real Power Above Configured High Limit', [41].Code := 45, [41].Desc := 'Reactive Power Below Configured Lo Limit', [42].Code := 46, [42].Desc := 'Reactive Power Above Configured Hi Limit', [43].Code := 47, [43].Desc := 'Apparent Power Below Configured Lo Limit', [44].Code := 48, [44].Desc := 'Apparent Power Above Configured Hi Limit', [45].Code := 49, [45].Desc := 'Power Line Frequency Out of Spec', [46].Code := 50, [46].Desc := 'Total Run Hours: PM is Required', [47].Code := 51, [47].Desc := 'Total Motor Starts: PM is Required', [48].Code := 52, [48].Desc := 'SCR Phase A Power Quality / Firing Fault', [49].Code := 53, [49].Desc := 'SCR Phase B Power Quality / Firing Fault', [50].Code := 54, [50].Desc := 'SCR Phase C Power Quality / Firing Fault', [51].Code := 55, [51].Desc := 'Power Quality V THD Out of Spec', [52].Code := 56, [52].Desc := 'Power Quality I THD Out of Spec', [53].Code := 57, [53].Desc := 'Configuration Changed', [54].Code := 58, [54].Desc := 'Excessive Ground Fault Current', [55].Code := 59, [55].Desc := 'Motor Overtemperature (from sensor)', [56].Code := 60, [56].Desc := 'Power Pole Overtemperature (from sensor)', [57].Code := 61, [57].Desc := 'SMC-50 I/O Configuration Fault', [58].Code := 62, [58].Desc := 'Push-to-Test (Test Trip) Fault', [59].Code := 63, [59].Desc := 'Lagging Power Factor below fault limit', [60].Code := 64,
        [60].Desc := 'Leading Power Factor below fault limit', [61].Code := 65, [61].Desc := 'Lagging Power Factor above fault limit', [62].Code := 66, [62].Desc := 'Leading Power Factor above fault limit', [63].Code := 67, [63].Desc := 'MVAR (Reactive Power) above fault limit', [64].Code := 68, [64].Desc := 'MVAR (Reactive Power) below fault limit', [65].Code := 69, [65].Desc := 'Replace SMC-50 Real-Time Clock Battery', [66].Code := 70, [66].Desc := 'Motor Locked Rotor fault');   // SMC-50 Smart Motor Controller Fault Code List
   SMCFlex_FaultCodeList : P_DescList[48] := ([0].Desc := 'Check starter manual for this fault code', [1].Code := 1, [1].Desc := 'Fault: Phase A Power / Line Lost', [2].Code := 2, [2].Desc := 'Fault: Phase B Power / Line Lost', [3].Code := 3, [3].Desc := 'Fault: Phase C Power / Line Lost', [4].Code := 4, [4].Desc := 'Fault: Shorted SCR for Phase A', [5].Code := 5, [5].Desc := 'Fault: Shorted SCR for Phase B', [6].Code := 6, [6].Desc := 'Fault: Shorted SCR for Phase C', [7].Code := 7, [7].Desc := 'Fault: Open Gate on SCR for Phase A', [8].Code := 8, [8].Desc := 'Fault: Open Gate on SCR for Phase B', [9].Code := 9, [9].Desc := 'Fault: Open Gate on SCR for Phase C', [10].Code := 10, [10].Desc := 'PTC (Temp Sensor) Power Pole Fault', [11].Code := 11, [11].Desc := 'SMCFlex SCR Overtemperature Fault', [12].Code := 12, [12].Desc := 'Motor Overtemperature Fault (or bad PTC)', [13].Code := 13, [13].Desc := 'Open Bypass Fault on Phase A', [14].Code := 14, [14].Desc := 'Open Bypass Fault on Phase B', [15].Code := 15, [15].Desc := 'Open Bypass Fault on Phase C', [16].Code := 16, [16].Desc := 'No Load on Phase A (broken wire?)', [17].Code := 17, [17].Desc := 'No Load on Phase B (broken wire?)', [18].Code := 18, [18].Desc := 'No Load on Phase C (broken wire?)', [19].Code := 19, [19].Desc := 'Line Unbalance Fault', [20].Code := 20, [20].Desc := 'Overvoltage Fault', [21].Code := 21, [21].Desc := 'Undervoltage Fault', [22].Code := 22, [22].Desc := 'Motor Overload Fault', [23].Code := 23, [23].Desc := 'Underload Fault (broken shaft?)', [24].Code := 24, [24].Desc := 'Jam Fault (Motor / Machine Stuck)', [25].Code := 25, [25].Desc := 'Stalled Motor Fault', [26].Code := 26, [26].Desc := 'Phase Reversal Fault', [27].Code := 27, [27].Desc := 'Comms Lost on Network Port 2 (HIM, etc.)', [28].Code := 28, [28].Desc := 'Comms Lost on Network Port 3 (HIM, etc.)', [29].Code := 29, [29].Desc := 'Comms Lost on Network Port 5 (Ethernet)', [30].Code := 30,
        [30].Desc := 'Network Port 2 Fault (HIM, etc.)', [31].Code := 31, [31].Desc := 'Network Port 3 Fault (HIM, etc.)', [32].Code := 32, [32].Desc := 'Net Port 5 Fault (Controller Comms/PROG)', [33].Code := 33, [33].Desc := 'Ground Fault', [34].Code := 34, [34].Desc := 'Starting too frequently', [35].Code := 35, [35].Desc := 'Phase A Power Lost', [36].Code := 36, [36].Desc := 'Phase B Power Lost', [37].Code := 37, [37].Desc := 'Phase C Power Lost', [38].Code := 38, [38].Desc := 'Hall Effect Sensor ID Fault', [39].Code := 39, [39].Desc := 'Nonvolatile Memory Error', [40].Code := 40, [40].Desc := 'Fault: No Load', [41].Code := 41, [41].Desc := 'Phase A Line Lost', [42].Code := 42, [42].Desc := 'Phase B Line Lost', [43].Code := 43, [43].Desc := 'Phase C Line Lost', [44].Code := 45, [44].Desc := '24 Volt Supply Lost', [45].Code := 46, [45].Desc := 'Voltage Control Lost', [46].Code := 48, [46].Desc := 'Input 1 Fault', [47].Code := 49, [47].Desc := 'Input 2 Fault');   // SMCFlex Soft Starter Fault Codes and Descriptions
END_VAR

PROGRAM Diagnostics   (* main routine L_CPU *)
VAR
   L_TaskInhibited : DINT[8] := ([0] := 1);   // GSV result: 'Task' class, 'InhibitTask' attribute
END_VAR

ROUTINE L_CPU   (* ladder *)
// Logix CPU Utilization, and checking for Inhibited Tasks
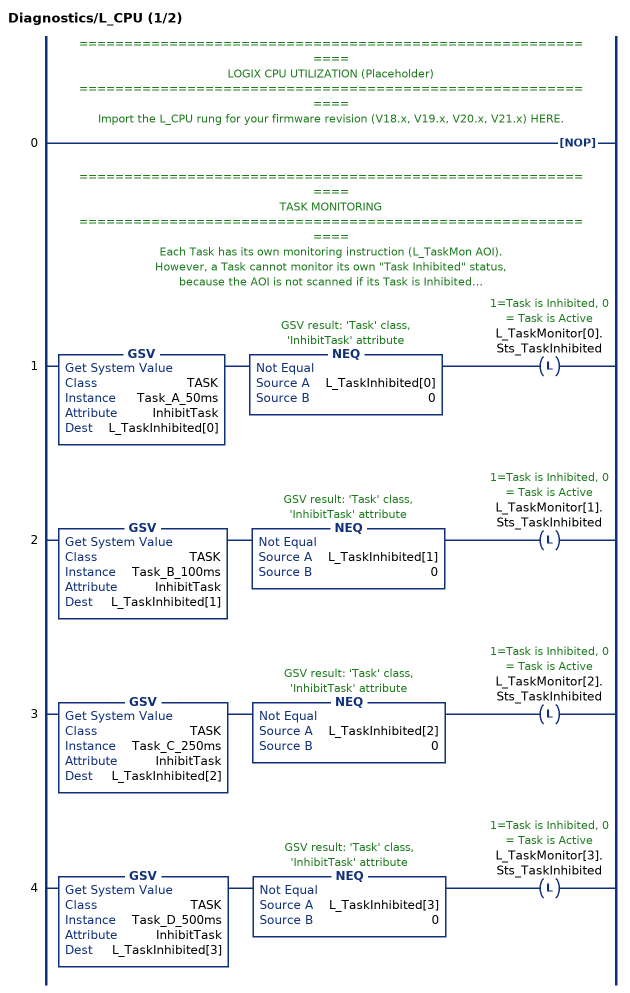
   // ============================================================
   // LOGIX CPU UTILIZATION (Placeholder)
   // ============================================================
   // Import the L_CPU rung for your firmware revision (V18.x, V19.x, V20.x, V21.x) HERE.
   0: NOP();
   // ============================================================
   // TASK MONITORING
   // ============================================================
   // Each Task has its own monitoring instruction (L_TaskMon AOI).
   // However, a Task cannot monitor its own "Task Inhibited" status,
   // because the AOI is not scanned if its Task is Inhibited!
   // So this small Task is used to monitor each of the other
   // controller Tasks and set the "TaskInhibited" Status
   // of those Tasks if they are set Inhibited.
   // Each rung below monitors the Inhibited status of
   // one of this controller's Tasks.
   1: GSV(TASK,Task_A_50ms,InhibitTask,L_TaskInhibited[0])NEQ(L_TaskInhibited[0],0)OTL(L_TaskMonitor[0].Sts_TaskInhibited);
   2: GSV(TASK,Task_B_100ms,InhibitTask,L_TaskInhibited[1])NEQ(L_TaskInhibited[1],0)OTL(L_TaskMonitor[1].Sts_TaskInhibited);
   3: GSV(TASK,Task_C_250ms,InhibitTask,L_TaskInhibited[2])NEQ(L_TaskInhibited[2],0)OTL(L_TaskMonitor[2].Sts_TaskInhibited);
   4: GSV(TASK,Task_D_500ms,InhibitTask,L_TaskInhibited[3])NEQ(L_TaskInhibited[3],0)OTL(L_TaskMonitor[3].Sts_TaskInhibited);
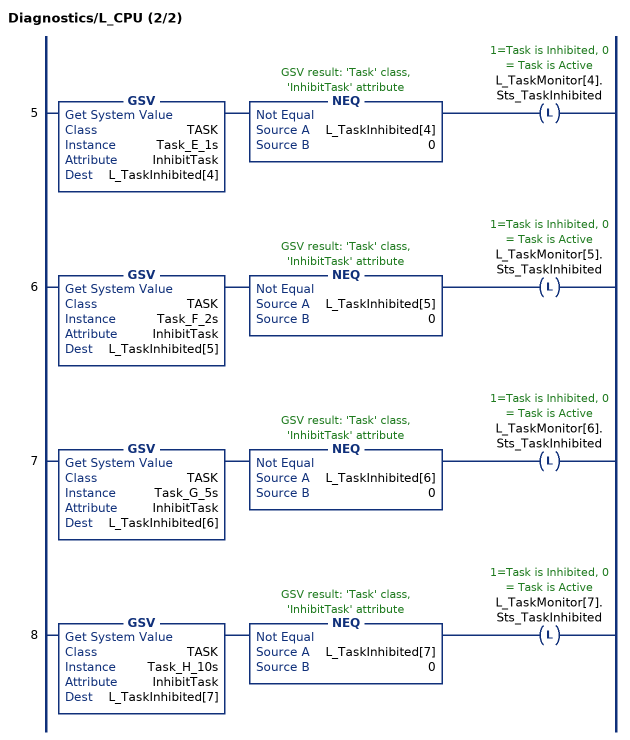
   5: GSV(TASK,Task_E_1s,InhibitTask,L_TaskInhibited[4])NEQ(L_TaskInhibited[4],0)OTL(L_TaskMonitor[4].Sts_TaskInhibited);
   6: GSV(TASK,Task_F_2s,InhibitTask,L_TaskInhibited[5])NEQ(L_TaskInhibited[5],0)OTL(L_TaskMonitor[5].Sts_TaskInhibited);
   7: GSV(TASK,Task_G_5s,InhibitTask,L_TaskInhibited[6])NEQ(L_TaskInhibited[6],0)OTL(L_TaskMonitor[6].Sts_TaskInhibited);
   8: GSV(TASK,Task_H_10s,InhibitTask,L_TaskInhibited[7])NEQ(L_TaskInhibited[7],0)OTL(L_TaskMonitor[7].Sts_TaskInhibited);
END_ROUTINE
END_PROGRAM

PROGRAM Tank1   (* main routine MainRoutine *)
VAR
   LC1_IOFault_Bor : FBD_BOOLEAN_OR; {access Read Only}
   LevelSim1 : JLB_FopdtSim := (cv := 30.00001, gain := 1.0, deadTime := 2.0, timeConst := 10.0, pv := 30.00001, pvLimitHigh := 100.0);
   LT1_PVBad_Bor : FBD_BOOLEAN_OR; {access Read Only}
   P1_ChanFault_Bor : FBD_BOOLEAN_OR; {access Read Only}
   P1_IOFault_Bor : FBD_BOOLEAN_OR; {access Read Only}
   P1_ModFault_Bor : FBD_BOOLEAN_OR; {access Read Only}
   P1_Out_Start : BOOL;   // Tag Descript - Output to Start Drive
   P1_Out_Stop : BOOL;   // Tag Descript - Output to Stop Drive
END_VAR
VAR_INPUT
   LC1_Out_CV_ChanFault : BOOL; {access Read Only}   // TagDescript - Control Variable Output Channel Fault
   LC1_Out_CV_ModFault : BOOL; {access Read Only}   // TagDescript - Control Variable Output Module Fault
   LT1_Inp_PV_ChanFault : BOOL; {access Read Only}   // TagDescript - Process Variable Input Channel Fault
   LT1_Inp_PV_ModFault : BOOL; {access Read Only}   // TagDescript - Process Variable Input Module Fault
   P1_Inp_Running : BOOL; {access Read Only}   // TagDescript - Runing Feedback Input
   P1_Inp_Running_ChanFault : BOOL; {access Read Only}   // TagDescript - Runing Feedback Input Channel Fault
   P1_Inp_Running_ModFault : BOOL; {access Read Only}   // TagDescript - Runing Feedback Input Module Fault
   P1_Inp_SpeedFdbk : REAL := 7561.6177; {access Read Only}   // TagDescript - Speed Feedback Input
   P1_Inp_SpeedFdbk_ChanFault : BOOL; {access Read Only}   // TagDescript - Speed Feedback Input Channel Fault
   P1_Inp_SpeedFdbk_ModFault : BOOL; {access Read Only}   // TagDescript - Speed Feedback Input Module Fault
   P1_Out_RunFwd_ChanFault : BOOL; {access Read Only}   // TagDescript - Run Forward Output Channel Fault
   P1_Out_RunFwd_ModFault : BOOL; {access Read Only}   // TagDescript - Run Forward Output Module Fault
   P1_Out_RunRev_ChanFault : BOOL; {access Read Only}   // TagDescript - Run Reverse Output Channel Fault
   P1_Out_RunRev_ModFault : BOOL; {access Read Only}   // TagDescript - Run Reverse Output Module Fault
   P1_Out_SpeedRef_ChanFault : BOOL; {access Read Only}   // TagDescript - Speed Reference Output Channel Fault
   P1_Out_SpeedRef_ModFault : BOOL; {access Read Only}   // TagDescript - Speed Reference Output Module Fault
END_VAR
VAR_OUTPUT
   P1_Out_SpeedRef : REAL := 7561.6177; {access Read Only}   // TagDescript - Speed Reference Output
END_VAR

ROUTINE LC1   (* function block diagram *)
// TagDescript
   SHEET 1   // PS_PID
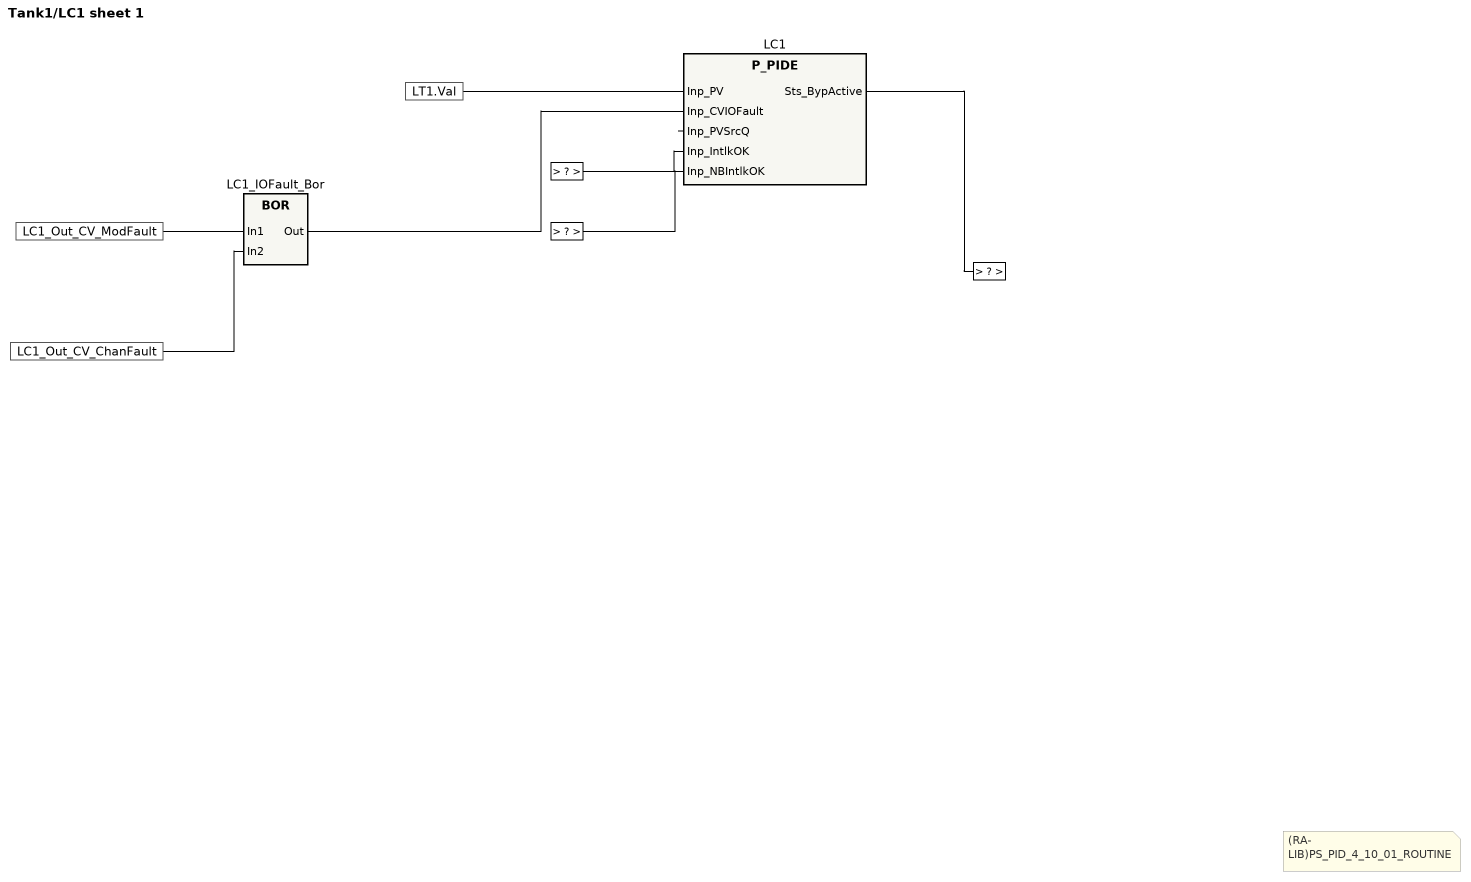
   // (RA-
   // LIB)PS_PID_4_10_01_ROUTINE
   LC1_IOFault_Bor : BOR(In1 := LC1_Out_CV_ModFault, In2 := LC1_Out_CV_ChanFault);
   LC1 : P_PIDE(Inp_PV := LT1.Val, Inp_CVIOFault := LC1_IOFault_Bor.Out, Inp_IntlkOK := WIRE(?), Inp_NBIntlkOK := WIRE(?));   // unwired pins: Inp_PVSrcQ
   WIRE(?) := LC1.Sts_BypActive;
   SHEET 2   // Interlocks
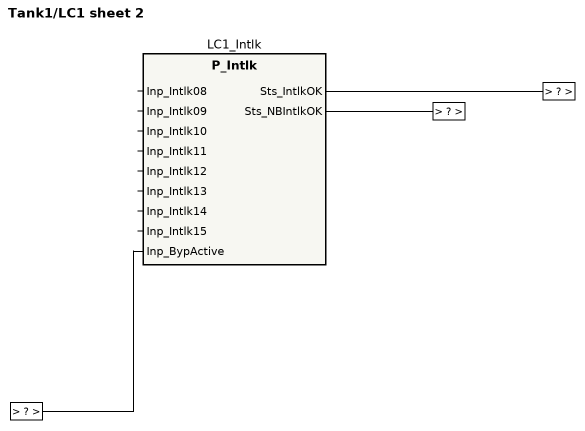
   LC1_Intlk : P_Intlk(Inp_BypActive := WIRE(?) {feedback});   // unwired pins: Inp_Intlk08 Inp_Intlk09 Inp_Intlk10 Inp_Intlk11 Inp_Intlk12 Inp_Intlk13 Inp_Intlk14 Inp_Intlk15
   WIRE(?) := LC1_Intlk.Sts_NBIntlkOK;
   WIRE(?) := LC1_Intlk.Sts_IntlkOK;
END_ROUTINE

ROUTINE LevelSim1   (* function block diagram *)
   SHEET 1
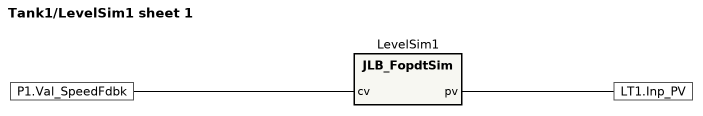
   LevelSim1 : JLB_FopdtSim(cv := P1.Val_SpeedFdbk);
   LT1.Inp_PV := LevelSim1.pv;
END_ROUTINE

ROUTINE LT1   (* function block diagram *)
// TagDescript
   SHEET 1   // PS_AIn
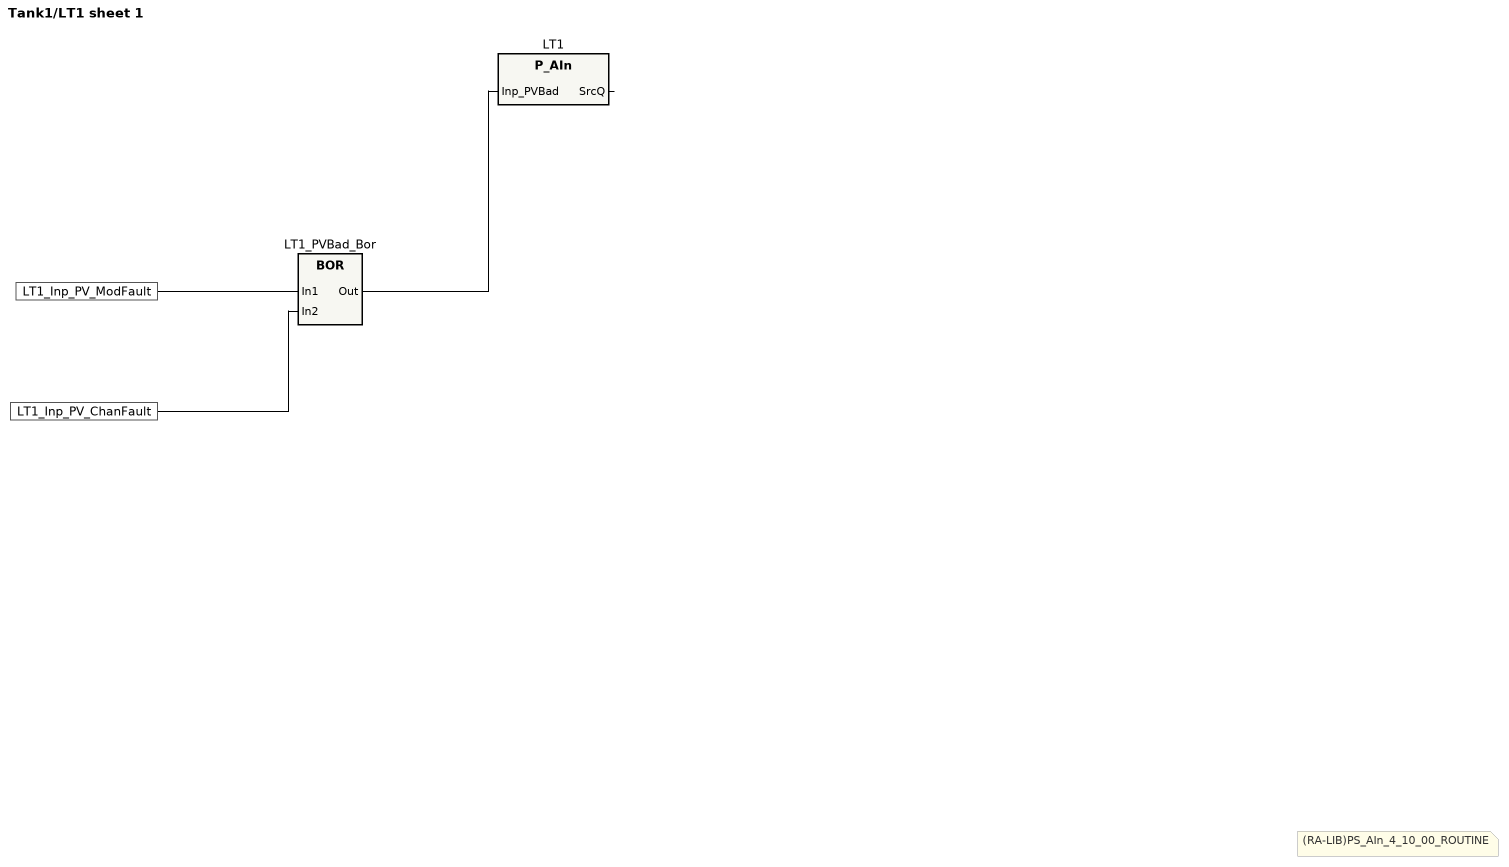
   // (RA-LIB)PS_AIn_4_10_00_ROUTINE
   LT1_PVBad_Bor : BOR(In1 := LT1_Inp_PV_ModFault, In2 := LT1_Inp_PV_ChanFault);
   LT1 : P_AIn(Inp_PVBad := LT1_PVBad_Bor.Out);   // unwired pins: SrcQ
END_ROUTINE

ROUTINE MainRoutine   (* ladder *)
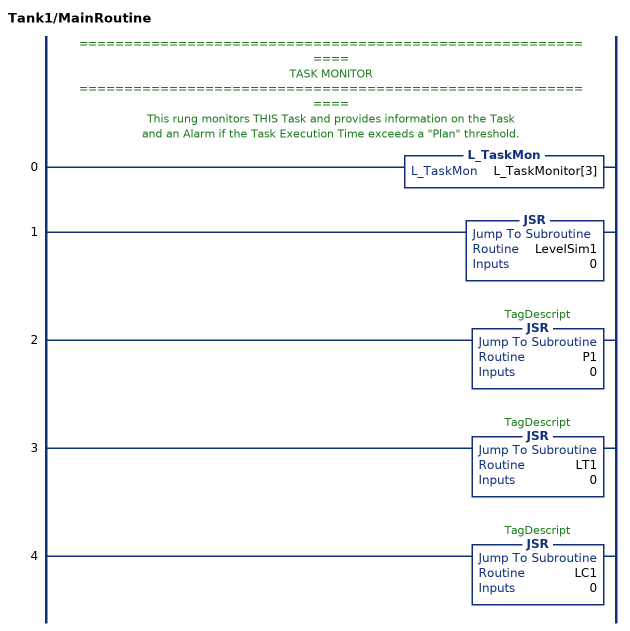
   // ============================================================
   // TASK MONITOR
   // ============================================================
   // This rung monitors THIS Task and provides information on the Task
   // and an Alarm if the Task Execution Time exceeds a "Plan" threshold.
   0: L_TaskMon(L_TaskMonitor[3]);
   1: JSR(LevelSim1,0);
   2: JSR(P1,0);
   3: JSR(LT1,0);
   4: JSR(LC1,0);
END_ROUTINE

ROUTINE P1   (* function block diagram *)
// TagDescript
   SHEET 1   // PS_VSD
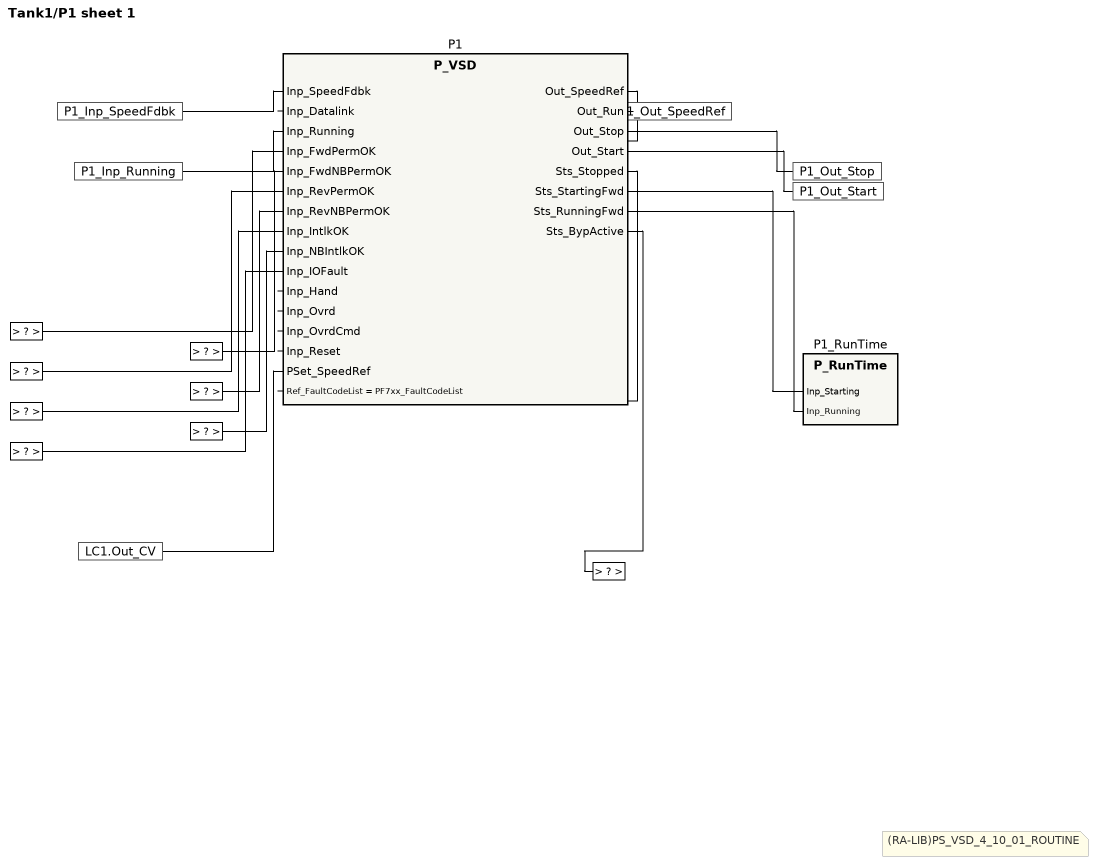
   // (RA-LIB)PS_VSD_4_10_01_ROUTINE
   P1 : P_VSD(Inp_SpeedFdbk := P1_Inp_SpeedFdbk, Inp_Running := P1_Inp_Running, Inp_FwdPermOK := WIRE(?), Inp_FwdNBPermOK := WIRE(?), Inp_RevPermOK := WIRE(?), Inp_RevNBPermOK := WIRE(?), Inp_IntlkOK := WIRE(?), Inp_NBIntlkOK := WIRE(?), Inp_IOFault := WIRE(?), PSet_SpeedRef := LC1.Out_CV, Ref_FaultCodeList := PF7xx_FaultCodeList);   // unwired pins: Inp_Datalink Inp_Hand Inp_Ovrd Inp_OvrdCmd Inp_Reset Out_Run
   WIRE(?) := P1.Sts_Stopped;
   WIRE(?) := P1.Sts_BypActive;
   P1_Out_SpeedRef := P1.Out_SpeedRef;
   P1_Out_Stop := P1.Out_Stop;
   P1_Out_Start := P1.Out_Start;
   P1_RunTime : P_RunTime(Inp_Starting := P1.Sts_StartingFwd, Inp_Running := P1.Sts_RunningFwd);
   SHEET 2   // Forward Permissives
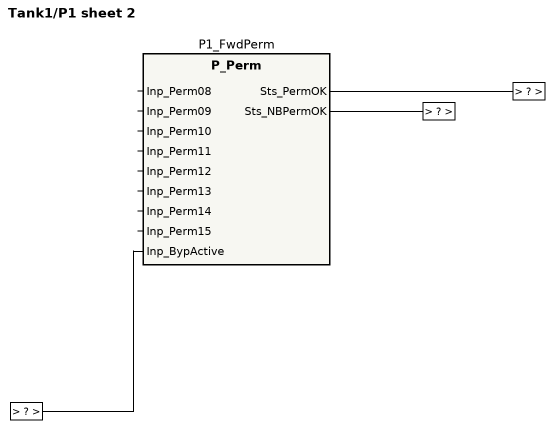
   P1_FwdPerm : P_Perm(Inp_BypActive := WIRE(?) {feedback});   // unwired pins: Inp_Perm08 Inp_Perm09 Inp_Perm10 Inp_Perm11 Inp_Perm12 Inp_Perm13 Inp_Perm14 Inp_Perm15
   WIRE(?) := P1_FwdPerm.Sts_NBPermOK;
   WIRE(?) := P1_FwdPerm.Sts_PermOK;
   SHEET 3   // Reverse Permissives
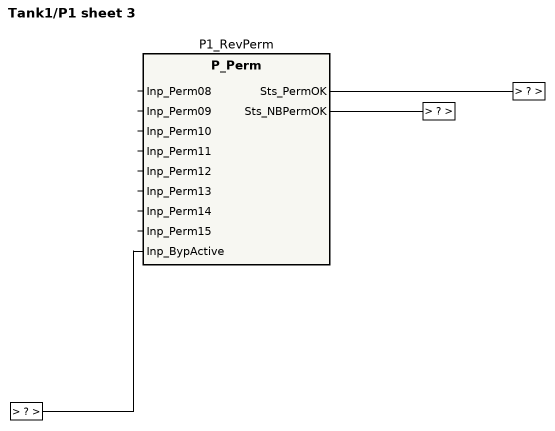
   P1_RevPerm : P_Perm(Inp_BypActive := WIRE(?) {feedback});   // unwired pins: Inp_Perm08 Inp_Perm09 Inp_Perm10 Inp_Perm11 Inp_Perm12 Inp_Perm13 Inp_Perm14 Inp_Perm15
   WIRE(?) := P1_RevPerm.Sts_NBPermOK;
   WIRE(?) := P1_RevPerm.Sts_PermOK;
   SHEET 4   // Interlocks
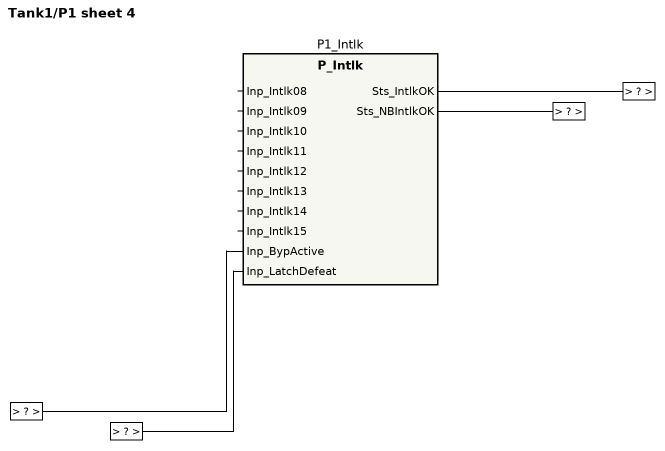
   P1_Intlk : P_Intlk(Inp_BypActive := WIRE(?) {feedback}, Inp_LatchDefeat := WIRE(?) {feedback});   // unwired pins: Inp_Intlk08 Inp_Intlk09 Inp_Intlk10 Inp_Intlk11 Inp_Intlk12 Inp_Intlk13 Inp_Intlk14 Inp_Intlk15
   WIRE(?) := P1_Intlk.Sts_NBIntlkOK;
   WIRE(?) := P1_Intlk.Sts_IntlkOK;
   SHEET 5   // IO Fault
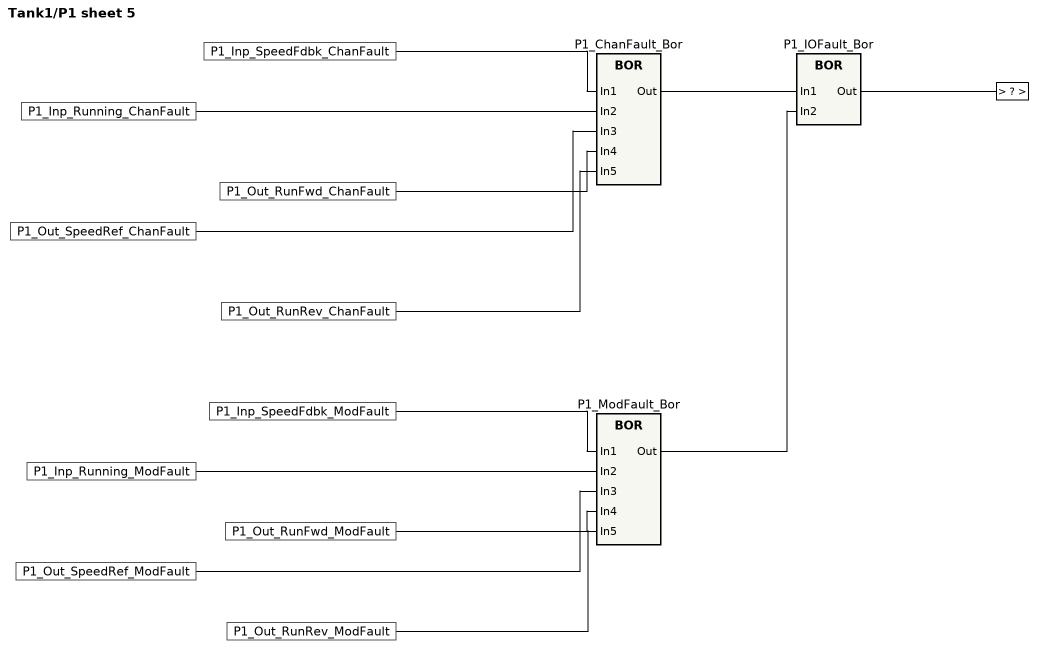
   P1_ChanFault_Bor : BOR(In1 := P1_Inp_SpeedFdbk_ChanFault, In2 := P1_Inp_Running_ChanFault, In3 := P1_Out_SpeedRef_ChanFault, In4 := P1_Out_RunFwd_ChanFault, In5 := P1_Out_RunRev_ChanFault);
   P1_ModFault_Bor : BOR(In1 := P1_Inp_SpeedFdbk_ModFault, In2 := P1_Inp_Running_ModFault, In3 := P1_Out_SpeedRef_ModFault, In4 := P1_Out_RunFwd_ModFault, In5 := P1_Out_RunRev_ModFault);
   P1_IOFault_Bor : BOR(In1 := P1_ChanFault_Bor.Out, In2 := P1_ModFault_Bor.Out);
   WIRE(?) := P1_IOFault_Bor.Out;
END_ROUTINE
END_PROGRAM

PROGRAM Task_A_MainProgram   (* main routine MainRoutine *)

ROUTINE MainRoutine   (* ladder *)
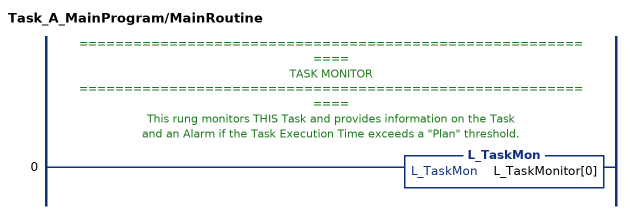
   // ============================================================
   // TASK MONITOR
   // ============================================================
   // This rung monitors THIS Task and provides information on the Task
   // and an Alarm if the Task Execution Time exceeds a "Plan" threshold.
   0: L_TaskMon(L_TaskMonitor[0]);
END_ROUTINE
END_PROGRAM

PROGRAM Task_B_MainProgram   (* main routine MainRoutine *)

ROUTINE MainRoutine   (* ladder *)
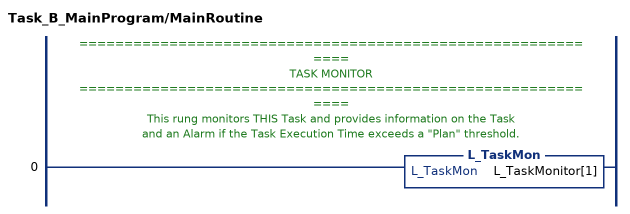
   // ============================================================
   // TASK MONITOR
   // ============================================================
   // This rung monitors THIS Task and provides information on the Task
   // and an Alarm if the Task Execution Time exceeds a "Plan" threshold.
   0: L_TaskMon(L_TaskMonitor[1]);
END_ROUTINE
END_PROGRAM

PROGRAM Task_C_MainProgram   (* main routine MainRoutine *)

ROUTINE MainRoutine   (* ladder *)
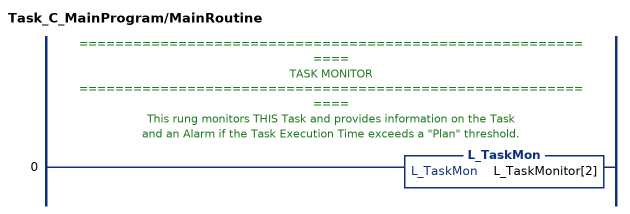
   // ============================================================
   // TASK MONITOR
   // ============================================================
   // This rung monitors THIS Task and provides information on the Task
   // and an Alarm if the Task Execution Time exceeds a "Plan" threshold.
   0: L_TaskMon(L_TaskMonitor[2]);
END_ROUTINE
END_PROGRAM

PROGRAM Task_E_MainProgram   (* main routine MainRoutine *)

ROUTINE MainRoutine   (* ladder *)
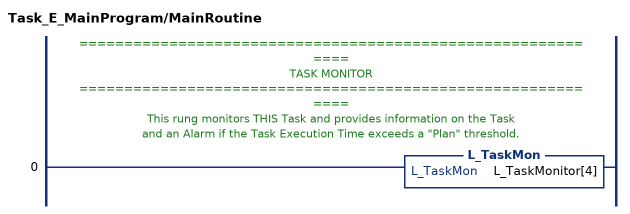
   // ============================================================
   // TASK MONITOR
   // ============================================================
   // This rung monitors THIS Task and provides information on the Task
   // and an Alarm if the Task Execution Time exceeds a "Plan" threshold.
   0: L_TaskMon(L_TaskMonitor[4]);
END_ROUTINE
END_PROGRAM

PROGRAM Task_F_MainProgram   (* main routine MainRoutine *)

ROUTINE MainRoutine   (* ladder *)
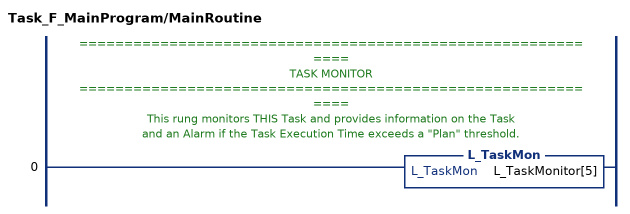
   // ============================================================
   // TASK MONITOR
   // ============================================================
   // This rung monitors THIS Task and provides information on the Task
   // and an Alarm if the Task Execution Time exceeds a "Plan" threshold.
   0: L_TaskMon(L_TaskMonitor[5]);
END_ROUTINE
END_PROGRAM

PROGRAM Task_G_MainProgram   (* main routine MainRoutine *)

ROUTINE MainRoutine   (* ladder *)
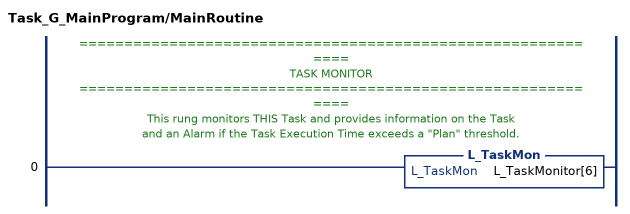
   // ============================================================
   // TASK MONITOR
   // ============================================================
   // This rung monitors THIS Task and provides information on the Task
   // and an Alarm if the Task Execution Time exceeds a "Plan" threshold.
   0: L_TaskMon(L_TaskMonitor[6]);
END_ROUTINE
END_PROGRAM
